// TIA Portal V17 export
// export: Created 2022-07-20T06:59:47.8919978Z, ExportSetting WithDefaults, DisplayName Totally Integrated Automation Portal, DisplayVersion V17, DisplayName TIA Portal Openness, DisplayVersion V17, DisplayName TIA Portal Version Control Interface, DisplayVersion V17, DisplayName SINAMICS Startdrive Advanced, DisplayVersion V17, DisplayName SINAMICS Startdrive G130, G150, S120, S150, SINAMICS MV, S210, DisplayVersion V17, DisplayName SINAMICS Startdrive G110M, G120, G120C, G120D, G120P, G115D, DisplayVersion V17, DisplayName STEP 7 Professional, DisplayVersion V17, DisplayName STEP 7 Safety, DisplayVersion V17, DisplayName WinCC Advanced, DisplayVersion V17
FUNCTION_BLOCK "FB10171_FanControl"   // FB10171, LAD
TITLE = FB10171_FanControl
{ S7_Optimized_Access := 'TRUE' }
AUTHOR : Jonathan
FAMILY : 1017_FAN
VERSION : 1.0
// Release note : 
// 1.0 - Feature developped
// stored: AutoNumber false, IsIECCheckEnabled false, IsRetainMemResEnabled false, MemoryReserve 100, SetENOAutomatically false, UDAEnableTagReadback false
   VAR_INPUT
      EnableModule : Bool;
      PowerOK : Bool;
      StartFanCommand : Bool;
      MaintainAfterStop : Bool;
      TimeToMaintainAfterStop : Time := T#1s;
   END_VAR
   VAR_OUTPUT
      ActivePowerRelay : Bool;
      StartFanSignal : Bool;
   END_VAR
   VAR
      TOF_MaintainAfterStop { S7_SetPoint := 'True'} : TOF_TIME;
   END_VAR
BEGIN

REGION Network 1: Active power relay
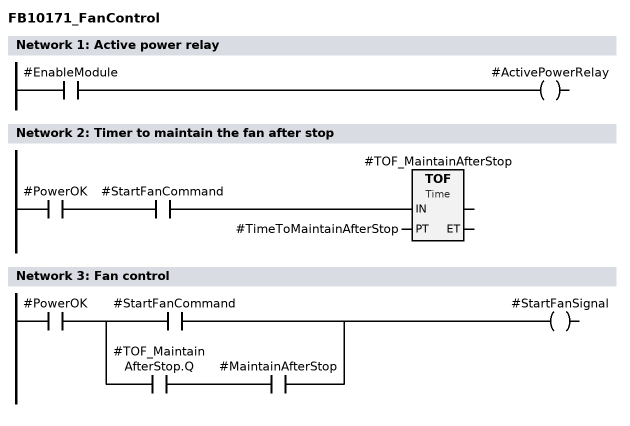
   RUNG wire#powerrail
      Contact( #EnableModule )
      Coil( #ActivePowerRelay )
   END_RUNG
   // the same network as SCL:
   #ActivePowerRelay := #EnableModule;
END_REGION

REGION Network 2: Timer to maintain the fan after stop
   RUNG wire#powerrail
      Contact( #PowerOK )
      Contact( #StartFanCommand )
      { S7_Templates := "time_type := Time" } #TOF_MaintainAfterStop.TOF(pt := #TimeToMaintainAfterStop, et =>)
   END_RUNG
   // the same network as SCL:
   #TOF_MaintainAfterStop(IN := #PowerOK AND #StartFanCommand, PT := #TimeToMaintainAfterStop);   // TOF
END_REGION

REGION Network 3: Fan control
   RUNG wire#powerrail
      Contact( #PowerOK )
      wire#w1
      Contact( #StartFanCommand )
      wire#w2
      Coil( #StartFanSignal )
   END_RUNG
   RUNG wire#w1
      Contact( #TOF_MaintainAfterStop.Q )
      Contact( #MaintainAfterStop )
   END_RUNG wire#w2
   // the same network as SCL:
   #StartFanSignal := #PowerOK AND (#StartFanCommand OR (#TOF_MaintainAfterStop.Q AND #MaintainAfterStop));
END_REGION
END_FUNCTION_BLOCK
